(* LS Electric XG5000 project: TEST-60 *)
(* PLC XEC-DN32H *)

PROGRAM NewProgram (* task: 스캔 프로그램 *)
VAR
    dDiffPressure : INT; (* 차압값 *)
    dHumidity : INT; (* 습도값 *)
    dTDS : DINT; (* TDS값 *)
    dWaterTemp : INT; (* 수온값 *)
    mAlarmDpTrip : BOOL; (* 차압 트립 알람 *)
    mAlarmDrainTO : BOOL; (* 배수 시간초과 알람 *)
    mAlarmRemote : BOOL; (* 원격 이상 알람 *)
    mAlarmReset AT %IX0.0.3 : BOOL; (* 알람 리셋 *)
    mAlarmSensor : BOOL; (* 센서 이상 알람 *)
    mAutoMode : BOOL; (* 자동 모드 *)
    mRemoteAlive : BOOL; (* 원격 통신 정상 *)
    mRemoteAuthOK : BOOL; (* 원격 인증 OK *)
    mRemoteDrainCmd : BOOL; (* 원격 배수 명령 *)
    mRemoteMode : BOOL; (* 원격 모드 *)
    mRemotePumpCmd : BOOL; (* 원격 펌프 명령 *)
    tBlower1Elapsed : TIME; (* 송풍기1 운전 경과시간 *)
    tBlower1RunET : TIME; (* 송풍기1 2시간 TON *)
    tBlower1RunIN : BOOL; (* 송풍기1 2시간 TON *)
    tBlower1RunPT : TIME; (* 송풍기1 2시간 TON *)
    tBlower1RunQ : BOOL; (* 송풍기1 2시간 TON *)
    tBlower2Elapsed : TIME; (* 송풍기2 운전 경과시간 *)
    tBlower2RunET : TIME; (* 송풍기2 2시간 TON *)
    tBlower2RunIN : BOOL; (* 송풍기2 2시간 TON *)
    tBlower2RunPT : TIME; (* 송풍기2 2시간 TON *)
    tBlower2RunQ : BOOL; (* 송풍기2 2시간 TON *)
    tDPConfirm : TON; (* 차압 확인 TON *)
    tDPElapsed : TIME; (* 차압 타이머 경과시간 *)
    tDrainElapsed : TIME; (* 배수 타이머 경과시간 *)
    tDrainLimit : TON; (* 배수 제한 TON *)
    xAutoDrainReq : BOOL; (* 자동 배수 요청 *)
    xAutoHeatReq : BOOL; (* 자동 히터 요청 *)
    xAutoPumpReq : BOOL; (* 자동 펌프 요청 *)
    xBlower1TimeUp : BOOL; (* 송풍기1 운전시간 완료 *)
    xBlower2TimeUp : BOOL; (* 송풍기2 운전시간 완료 *)
    xBlowerSelect : BOOL; (* 송풍기 선택 FALSE=1호기 TRUE=2호기 *)
    xDPDone : BOOL; (* 차압 타이머 완료 *)
    xDPHigh : BOOL; (* 차압 150 이상 조건 *)
    xDpTripLatched : BOOL; (* 차압 트립 래치 *)
    xDrainDone : BOOL; (* 배수 타이머 완료 *)
    xDrainLock : BOOL; (* 배수 시간초과 락 *)
    xDrainReqFinal : BOOL; (* 최종 배수 요청 *)
    xDrainValveRaw : BOOL; (* 배수밸브 임시 조건 *)
    xEStop AT %IX0.0.2 : BOOL; (* 비상정지 *)
    xPumpReqFinal : BOOL; (* 최종 펌프 요청 *)
    xRemotePermit : BOOL; (* 원격 허가 *)
    xResetPermit : BOOL; (* 리셋 허가 조건 *)
    xRunCmd : BOOL; (* 운전 래치 *)
    xSensorFault : BOOL; (* 센서 이상 *)
    xStartBtn AT %IX0.0.0 : BOOL; (* 시삭버튼 *)
    xStopBtn AT %IX0.0.1 : BOOL; (* 정지 버튼 *)
    xSystemOK : BOOL; (* 시스템 운전 가능 *)
    yAlarmOut AT %QX0.0.5 : BOOL; (* 공통 알람 출력 *)
    yBlower AT %QX0.0.0 : BOOL; (* 송풍기 출력 *)
    yDrainValve AT %QX0.0.2 : BOOL; (* 배수밸브 출력 *)
    yHeater AT %QX0.0.4 : BOOL; (* 히터 출력 *)
    yMakeupValve AT %QX0.0.3 : BOOL; (* 보급밸브 출력 *)
    yPump AT %QX0.0.1 : BOOL; (* 펌프 출력 *)
END_VAR
xSensorFault := (dDiffPressure > INT#500)
    OR (dTDS > DINT#50000)
    OR (dHumidity > INT#100)
    OR (dWaterTemp > INT#80);

mAlarmSensor := xSensorFault;


xRemotePermit := mRemoteMode AND mRemoteAuthOK AND mRemoteAlive;

mAlarmRemote := mRemoteMode AND NOT xRemotePermit;


xDPHigh := dDiffPressure >= INT#150;

tDPConfirm(IN:=xDPHigh, PT:=T#2S, Q=>xDPDone, ET=>tDPElapsed);


xResetPermit := mAlarmReset AND NOT xEStop AND (dDiffPressure <= INT#140);


xDpTripLatched := (xDpTripLatched OR xDPDone) AND NOT xResetPermit;

mAlarmDpTrip := xDpTripLatched;


xRunCmd := (xRunCmd OR (xStartBtn AND NOT xEStop AND NOT xDpTripLatched))
    AND NOT xStopBtn
    AND NOT xEStop
    AND NOT xDpTripLatched;


xAutoDrainReq := (xAutoDrainReq OR (dTDS >= DINT#4000))
    AND NOT (dTDS <= DINT#3500);


xAutoPumpReq := (xAutoPumpReq OR (dHumidity <= INT#70))
    AND NOT (dHumidity >= INT#80);


xAutoHeatReq := (xAutoHeatReq OR (dWaterTemp <= INT#5))
    AND NOT (dWaterTemp >= INT#8);


xSystemOK := xRunCmd
    AND NOT xEStop
    AND NOT xDpTripLatched
    AND NOT xSensorFault;


xPumpReqFinal := (xRemotePermit AND mRemotePumpCmd)
    OR ((NOT xRemotePermit) AND mAutoMode AND xAutoPumpReq);


xDrainReqFinal := (xRemotePermit AND mRemoteDrainCmd)
    OR ((NOT xRemotePermit) AND mAutoMode AND xAutoDrainReq);


xDrainValveRaw := xSystemOK
    AND NOT xDrainLock
    AND xDrainReqFinal;


tDrainLimit(IN:=xDrainValveRaw, PT:=T#120S, Q=>xDrainDone, ET=>tDrainElapsed);


xDrainLock := (xDrainLock OR xDrainDone) AND NOT xResetPermit;

mAlarmDrainTO := xDrainLock;


tBlower1Run(IN:=xSystemOK AND NOT xBlowerSelect, PT:=T#7200S, Q=>xBlower1TimeUp, ET=>tBlower1Elapsed);

tBlower2Run(IN:=xSystemOK AND xBlowerSelect, PT:=T#7200S, Q=>xBlower2TimeUp, ET=>tBlower2Elapsed);


IF xBlower1TimeUp THEN
    xBlowerSelect := TRUE;
END_IF;

IF xBlower2TimeUp THEN
    xBlowerSelect := FALSE;
END_IF;

yBlower1 := xSystemOK AND NOT xBlowerSelect;

yBlower2 := xSystemOK AND xBlowerSelect;

yHeater := xSystemOK AND xAutoHeatReq;

yPump := xSystemOK AND xPumpReqFinal;

yDrainValve := xSystemOK
    AND NOT xDrainLock
    AND xDrainReqFinal;

yMakeupValve := xSystemOK
    AND NOT xDrainLock
    AND xDrainReqFinal;

yAlarmOut := xEStop
    OR mAlarmDpTrip
    OR mAlarmDrainTO
    OR mAlarmSensor
    OR mAlarmRemote;
END_PROGRAM